{attribute 'linkalways'} 
{attribute 'no_explicit_call' := 'This FB is a CLASS and must be accessed using methods or properties'}
{attribute 'enable_dynamic_creation'}
FUNCTION_BLOCK State IMPLEMENTS I_State
VAR
	_name : STRING;
END_VAR

METHOD Execute
END_METHOD

METHOD FB_init : BOOL
VAR_INPUT
	bInitRetains : BOOL; // if TRUE, the retain variables are initialized (warm start / cold start)
	bInCopyCode : BOOL;  // if TRUE, the instance afterwards gets moved into the copy code (online change)
	name : STRING;
END_VAR
_name := name;
END_METHOD

PROPERTY Name : STRING
GET
Name := _name;
END_GET
END_PROPERTY

METHOD OnEntry
END_METHOD

METHOD OnExit
END_METHOD

END_FUNCTION_BLOCK

(* stored: Version 1.1.0.1, ProductVersion 3.1.4024.12
   POU State: Id {80ad0bd5-49ad-0ee9-008f-f7949e0ce51f}, SpecialFunc None
   Method Execute: Id {debb21bd-04af-0171-3ce7-4f63e3de10b8}
   Method FB_init: Id {ca57a798-fce6-0d46-0659-f20420d8fe5a}
   Property Name: Id {9d326383-68d4-0c07-3410-82ebca9c5e80}
   Get Get: Id {c0646918-1e60-0d15-2d86-d7d578e7a8db}
   Method OnEntry: Id {82854e59-864e-0f50-0bb9-4d65044e3598}
   Method OnExit: Id {3f50052d-45d0-0488-3160-4a4d7f734745} *)
